{attribute 'GeneratedUsingTerminal: EL3773-0000-0021'}
{attribute addProperty BoxType "EL3773-0000-0021"}
{attribute addProperty Id "I2_StatusAT %I*I2_Status_DC9039207"}
{attribute addProperty CRC "4239878219"}
{attribute addProperty Size "7"}
TYPE L2_Current_Status_FCB7684B EXTENDS TcoIo.InputBase_8311D824 :
STRUCT
	{attribute addProperty Name "I2_Status"}
	I2_Status AT %I* : I2_Status_DC903920;
END_STRUCT
END_TYPE

(* stored: Version 1.2.0.0, ProductVersion 3.1.4024.11
   DUT L2_Current_Status_FCB7684B: Id {f40d3169-124d-4012-ad92-58e88ccaa11d} *)
